# EPICS substitutions: hyrel3dApp/Db/asynRecord.substitutions
file asynRecord.template
{
	pattern { P		 , R		    , PORT	, ADDR , OMAX , IMAX }
		{ XF:11ID-M3 , "{Hyrel:1}"	, HYREL	, 0	   , 0	  , 0	}
}
